(* PLC project Programme MGS_2-07_refactorJOY.project, CODESYS CODESYS V3.5 SP19 Patch 1 *)
(* stored: creationDateTime 2026-06-29T23:37:38.689101, modificationDateTime 2026-06-29T22:49:33.424 *)

FUNCTION_BLOCK FB_Safety
  VAR_INPUT
    Enable : BOOL;  (* Active la surveillance *)
    Reset : BOOL;  (* Front d'acquittement des défauts *)
    EStopArmed : BOOL;  (* Entrée TOR fail-safe (TRUE = OK, FALSE = Déclenché) *)
    CanOnline : BOOL;  (* Trame com active (TRUE = OK) *)
    CanOperational : BOOL;  (* Nœud en marche (TRUE = OK) *)
    EthercatOk : BOOL;  (* Bus EtherCAT sain (TRUE = OK) *)
  END_VAR
  VAR_OUTPUT
    Ready : BOOL;  (* Logique de sécurité opérationnelle *)
    SafeStop : BOOL;  (* Ordre d'arrêt absolu (TRUE = STOP IMMÉDIAT) *)
    SafetyOk : BOOL;  (* Feu vert global (TRUE = Autorisation de bouger) *)
    Error : BOOL;  (* Présence anomalie sécurité *)
    ErrorId : WORD;  (* Code bitfield de la cause du déclenchement *)
  END_VAR

            // 🛑 1. GATE AUTOMATE
IF NOT Enable THEN
    Ready := FALSE;
    SafeStop := TRUE;             // Sécurité par défaut : arrêt forcé
    SafetyOk := FALSE;
    RETURN;
END_IF;

Ready := TRUE;

// 🔑 2. RESET DÉFAUTS
IF Reset AND Error THEN
    Error := FALSE;
    ErrorId := 16#0000;
END_IF;

// 🛡️ 3. LOGIQUE FAIL-SAFE (Perte de signal = Danger)
IF NOT EStopArmed THEN
    ErrorId := 16#0001;           // Code : Arrêt d'urgence activé
ELSIF NOT CanOnline OR NOT CanOperational THEN
    ErrorId := 16#0002;           // Code : Liaison Joystick perdue
ELSIF NOT EthercatOk THEN
    ErrorId := 16#0004;           // Code : Bus EtherCAT en faute
END_IF;

// 📤 4. ARBITRAGE DES SORTIES TRANSVERSES
Error := (ErrorId <> 16#0000);

// SafeStop est l'actionneur logiciel (TRUE = On coupe tout)
SafeStop := Error;

// SafetyOk est le feu vert (TRUE = Tout est sain)
SafetyOk := NOT Error;
          
END_FUNCTION_BLOCK
